FUNCTION_BLOCK CompositeFB1
  (* Standard: 61499-2 *)
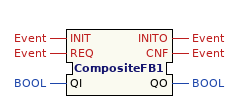
  EVENT_INPUT
    INIT;
    REQ;
  END_EVENT
  EVENT_OUTPUT
    INITO;
    CNF;
  END_EVENT
  VAR_INPUT
    QI : BOOL;
  END_VAR
  VAR_OUTPUT
    QO : BOOL;
  END_VAR
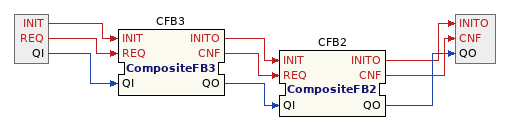
  FBS
    CFB2 : CompositeFB2;
    CFB3 : CompositeFB3;
  END_FBS
  EVENT_CONNECTIONS
    INIT TO CFB3.INIT;
    REQ TO CFB3.REQ;
    CFB3.INITO TO CFB2.INIT;
    CFB3.CNF TO CFB2.REQ;
    CFB2.INITO TO INITO;
    CFB2.CNF TO CNF;
  END_CONNECTIONS
  DATA_CONNECTIONS
    QI TO CFB3.QI;
    CFB3.QO TO CFB2.QI;
    CFB2.QO TO QO;
  END_CONNECTIONS
END_FUNCTION_BLOCK
